SUBAPPLICATION Automatik_Toggle_Button (* Automatik/Hand-Umschalter: 1 VT-Button (latched Toggle) -> Automatik-Zustand als AX-Plug (AUTOMATIK) + dessen Inverses (AX_MAN, fuer PID-Regler MAN-Eingang) + lokaler Publish (ID_AUTOMATIK_STATE_WRITE) fuer VT-Status/Web-Dashboard. Wiederverwendbar fuer jede Automatik-Funktion (Oelkuehler, Aufnahme, ...). *)
  (* Standard: 61499-2; Description: Copyright (c) 2026 Meisterschulen am Ostbahnhof This program and the accompanying materials are made available under the terms of the Eclipse Public License 2.0 which is available at https://www.eclipse.org/legal/epl-2.0/ SPDX-License-Identifier: EPL-2.0 *)
  (* Version 1.12, 2026-09-29, Franz Höpfinger, Meisterschulen am Ostbahnhof, Franz: AUTOMATIK_TOGGLED war falsch benannt/gefiltert - feuerte bei JEDEM Klick, auch beim Ausschalten. Umbenannt in AUTOMATIK_SET_FROM_VT und per neuem E_SWITCH (G=E_T_FF_Automatik.Q VOR dem Klick, ueber AX_SPLIT_4_Automatik auf AX_SPLIT_5 erweitert) gefiltert: EO0 (G=0, AUS->EIN) feuert AUTOMATIK_SET_FROM_VT UND E_T_FF_Automatik.S, EO1 (G=1, EIN->AUS) feuert nur E_T_FF_Automatik.R. CLK jetzt unbenutzt (ersatzlos, S/R decken beide Richtungen ab). *)
  (* Version 1.11, 2026-09-29, Franz Höpfinger, Meisterschulen am Ostbahnhof, Franz: 'Button_Softkey_Aux_IE mergt bereits intern, man kann das Merge rausnehmen' - E_MERGE_Toggle entfernt (Button_Automatik_Toggle ist seit Franz' eigenem Umbau bereits MyLib::sys::Button_Softkey_Aux_IE, das Button/Softkey/Aux selbst zu einem IND zusammenfuehrt; der separate TOGGLE-SubAppEventInput war ohnehin schon unbenutzt/entfernt). Button_Automatik_Toggle.IND geht jetzt direkt auf AX_E_PERMIT_2.EI2. Neuer SubAppEventOutput AUTOMATIK_TOGGLED (von AX_E_PERMIT_2.EO2, also PERMIT-gefiltert) - feuert bei jedem Klick, der die Automatik tatsaechlich toggelt (Button/Softkey/Aux gleichermassen). Fuer Bunker_Ernte_Automatik.SUB: SET soll durch den Display-Klick kommen, nicht durch das FORCE_ON-Echo (Franz-Diagnose: B05-Flattern -> Bunker_Komplett_Absenken.FORCE_ON_OUT -> Befuellautomatik AUTOMATIK-Republish -> Bunker_Ernte_Automatik.ACTIVE wird ueber dieselbe B05-Flanke sofort wieder gesetzt UND resettet, Latch flackert). *)
  (* Version 1.9, 2026-09-27, Franz Höpfinger, Meisterschulen am Ostbahnhof, Franz: 'soll das GESAMTE AN/Aus gaten, beim Uebergang 1->0 einmalig RESET, sonst wirkt es wie ein AX_PERMIT'. Neuer Socket PERMIT (AX). AX_SPLIT_2 speist AX_E_PERMIT_2 (gated FORCE_ON + Button_Automatik_Toggle.IND durch, nur wenn PERMIT=TRUE) und einen neuen AX_F_TRIG (fallende Flanke auf PERMIT -> E_T_FF_Automatik.R). *)
  (* Version 1.8, 2026-09-27, Franz Höpfinger, Meisterschulen am Ostbahnhof, Franz: 'FORCE_ON und FORCE_OFF sollten EVENTS sein, alles andere macht keinen Sinn' - von AX-Sockets (mit internem AX_R_TRIG zur Flankenerkennung) auf echte SubAppEventInputs umgestellt, direkt auf E_T_FF_Automatik.S/.R verdrahtet (wie das bereits bestehende AUS-Event). AX_R_TRIG_ForceOn/_ForceOff entfallen ersatzlos. Aufrufer mit pegelbasierten Quellen (Subscribes, ODER/UND-Verknuepfungen) muessen jetzt selbst die Flankenerkennung vor der Event-Verbindung liefern - siehe Befuellautomatik.SUB/Aufnahme_Automatik.SUB. *)
  (* Version 1.7, 2026-09-20, Franz Höpfinger, Meisterschulen am Ostbahnhof, Bugfix: seit v1.6 (Button_IE statt Softkey_IE, Latchable=0) kommt der Klick zwar an, aber der Button zeigte den AUTOMATIK-Zustand nicht mehr an - bei Latchable=1 hatte das VT dieses Feedback bisher selbst uebernommen (eigene Latched-Optik), das entfaellt jetzt. Neue SubApp Background_Automatik (GreenWhiteBackground3_AX, faerbt Button UND AUX gruen/weiss) ergaenzt, AX_SPLIT_3_Automatik auf AX_SPLIT_4_Automatik erweitert (4. Ausgang -> Background_Automatik.DI1). *)
  (* Version 1.6, 2026-09-20, Franz Höpfinger, Meisterschulen am Ostbahnhof, Bugfix: Button_Automatik_Toggle nutzte Softkey_Aux_IE (Softkey_IE) mit einer echten VT-Button-Object-ID (CButton, z.B. Button_Aufnahme_Geschwindigkeitsregelung_EinAus) - Softkey_IE empfaengt aber keine Button-Activation-Message, der Toggle-Klick kam nie an, AUTOMATIK blieb dauerhaft auf bDefaultAutomatik stehen. Neuer Baustein Button_Aux_IE (Button_IE statt Softkey_IE) - der VT-Button muss dafuer non-latching sein (Latchable=0), wird von Franz direkt im Pool umgestellt. *)
  (* Version 1.5, 2026-09-16, Franz Höpfinger, Meisterschulen am Ostbahnhof, Event-Input RESET in AUS umbenannt (Franz: 'der Eingang soll AUS heissen') - Namenskonsistenz mit AX_SoftkeyToggle_RS_TO_AX(_BG_PUBLISH)/Baender_Individual_Toggle/Baender_EinAus/Aufnahme_Automatik/Ernteseite_Antriebe. *)
  (* Version 1.4, 2026-09-16, Franz Höpfinger, Meisterschulen am Ostbahnhof, Event-Input RESET ergaenzt (rein additiv, zusaetzlich zum bestehenden Reset.IND-Pfad auf E_T_FF_Automatik.R verdrahtet) - fuer einen zentral gelesenen, gemeinsamen SoftKey (z.B. 'Alles Aus'), der mehrere Automatik-Instanzen gleichzeitig per Event zuruecksetzen soll. *)
  (* Version 1.3, 2026-09-15, Franz Höpfinger, Meisterschulen am Ostbahnhof, AUX-Unterstuetzung ergaenzt: Button_Automatik_Toggle von isobus::UT::io::Button::Button_IE (nur SoftKey) auf MyLib::sys::Softkey_Aux_IE (SoftKey ODER AUX) umgestellt, neuer optionaler InputVar u16ObjIdA_Automatik_Toggle (Default ID_NULL) - etabliertes Muster aus AX_SoftkeyToggle_RS_TO_AX.SUB uebernommen. Rein additiv, bestehende Instanzen ohne AUX-Wert funktionieren unveraendert. *)
  (* Version 1.2, 2026-09-13, Franz Höpfinger, Meisterschulen am Ostbahnhof, FORCE_ON/FORCE_OFF Sockets (AX) ergaenzt - rein FB-interne (nicht VT-Objekt-basierte) Gegenstuecke zum bestehenden VT-Reset, je per AX_R_TRIG (steigende Flanke) auf E_T_FF_Automatik.S bzw. .R. Fuer Automatik-zu-Automatik-Verknuepfungen (z.B. Befuellautomatik EIN schaltet Bunker-Ernte-Automatik automatisch mit ein; ein Kollisionsschutz schaltet eine Automatik hart aus) - rein additiv, bestehende Instanzen unveraendert nutzbar. *)
  (* Version 1.1, 2026-09-13, Franz Höpfinger, Meisterschulen am Ostbahnhof, Reset-Eingang ergaenzt (u16ObjId_RESET/u16ObjIdA_RESET/ID_RESET_METHOD -> MyLib::sys::Softkey_Aux_Method_IE -> E_T_FF_Automatik.R), analog AX_SoftkeyToggle_RS_TO_AX - fuer eine globale Sammel-AUS-Taste (SoftKey_AUS), die die Automatik hart auf Hand/AUS zurueckschalten muss (KVE14 Funktionen und Bedingungen Zeile 19, 'Aufnahme, Saege und Baender AUS'). *)
  (* Version 1.0, 2026-09-12, Franz Höpfinger, Meisterschulen am Ostbahnhof, initial implementation - aus Aufnahme_Automatik.SUB herausgeloest (Button_Automatik_Toggle/E_T_FF_Automatik/AX_SPLIT_3_Automatik/AX_NOT_Man/AX_PUBLISH_Automatik), generisch wiederverwendbar. *)
  PACKAGE MyLib::sys;
  IMPORT isobus::UT::Q::const::IDs::ID_NULL;
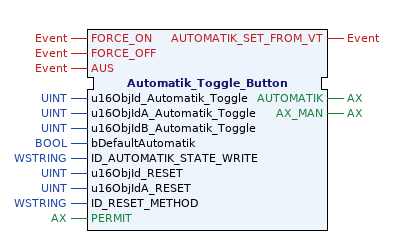
  EVENT_INPUT
    FORCE_ON; (* Schaltet die Automatik hart EIN (z.B. von einer anderen, uebergeordneten Automatik oder einem Methodenaufruf). Unverdrahtet lassen, wenn nicht gebraucht. *)
    FORCE_OFF; (* Schaltet die Automatik hart AUS (z.B. von einem Kollisionsschutz-Methodenaufruf). Unverdrahtet lassen, wenn nicht gebraucht. *)
    AUS; (* Reset hart auf Hand/AUS, von aussen als Event (z.B. 1 zentral gelesener gemeinsamer SoftKey) - zusaetzlich zum eigenen u16ObjId_RESET/u16ObjIdA_RESET/ID_RESET_METHOD-Pfad. Unverdrahtet lassen, wenn nicht gebraucht. *)
  END_EVENT
  EVENT_OUTPUT
    AUTOMATIK_SET_FROM_VT; (* Feuert nur beim Klick (Button/Softkey/Aux, PERMIT-gefiltert), der die Automatik von AUS auf EIN schaltet (per E_SWITCH auf dem Q-Zustand VOR dem Klick gefiltert - ein Klick der AUS schaltet feuert das NICHT). Echter Display-Klick-Event, kein Zustands-Level/Republish. *)
  END_EVENT
  VAR_INPUT
    u16ObjId_Automatik_Toggle : UINT := ID_NULL; (* Object ID VT-Softkey (Automatik/Hand-Umschalter) *)
    u16ObjIdA_Automatik_Toggle : UINT := ID_NULL; (* Object ID AuxFunction2 (Joystick), gleichberechtigt zum VT-Button - optional, ID_NULL wenn kein AUX gebraucht wird *)
    u16ObjIdB_Automatik_Toggle : UINT; (* Object ID VT-Button (Automatik/Hand-Umschalter) *)
    bDefaultAutomatik : BOOL := FALSE; (* Automatik-Zustand beim Start *)
    ID_AUTOMATIK_STATE_WRITE : WSTRING; (* Lokale Publish-Adresse (BOOL, ACTION=WRITE) fuer den Automatik-Ein/Aus-Zustand - Status-Text auf der VT + Web-Client/Dashboard *)
    u16ObjId_RESET : UINT := ID_NULL; (* Object ID Softkey 'Alles Aus' (Reset, hart auf Hand/AUS) - z.B. SoftKey_AUS *)
    u16ObjIdA_RESET : UINT := ID_NULL; (* Object ID AuxFunction2 (Joystick) fuer den Reset - gleichberechtigt zum Softkey 'Alles Aus' *)
    ID_RESET_METHOD : WSTRING; (* Lokale Methodenadresse (ACTION=CREATE_METHOD) fuer den argumentlosen Reset-Trigger (hart auf Hand/AUS) - wird von Web-Client UND OPC-Dashboard aufgerufen *)
  END_VAR
  SOCKETS
    PERMIT : adapter::types::unidirectional::AX;
  END_SOCKETS
  PLUGS
    AUTOMATIK : adapter::types::unidirectional::AX; (* Automatik aktiv (roh, z.B. fuer eine Freigabe-UND-Verknuepfung) *)
    AX_MAN : adapter::types::unidirectional::AX; (* NICHT Automatik aktiv (fuer PID-Regler MAN-Eingang) *)
  END_PLUGS
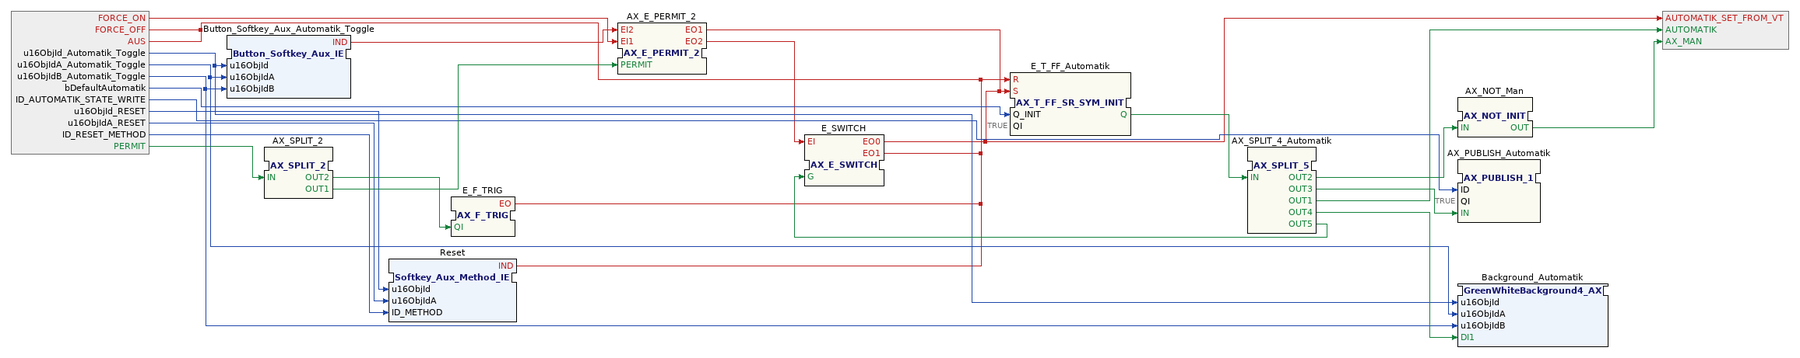
  FBS
    E_T_FF_Automatik : adapter::events::unidirectional::AX_T_FF_SR_SYM_INIT(QI := TRUE);
    AX_SPLIT_4_Automatik : adapter::events::unidirectional::AX_SPLIT_5;
    AX_NOT_Man : adapter::booleanOperators::AX_NOT_INIT;
    AX_PUBLISH_Automatik : adapter::net::AX_PUBLISH_1(QI := TRUE);
    AX_E_PERMIT_2 : adapter::events::unidirectional::AX_E_PERMIT_2;
    AX_SPLIT_2 : adapter::events::unidirectional::AX_SPLIT_2;
    E_F_TRIG : adapter::events::unidirectional::AX_F_TRIG;
    E_SWITCH : adapter::events::unidirectional::AX_E_SWITCH;
  END_FBS
  SUBAPPS
    Button_Softkey_Aux_Automatik_Toggle : MyLib::sys::Button_Softkey_Aux_IE;
    Background_Automatik : MyLib::sys::GreenWhiteBackground4_AX;
    Reset : MyLib::sys::Softkey_Aux_Method_IE;
  END_SUBAPPS
  EVENT_CONNECTIONS
    Button_Softkey_Aux_Automatik_Toggle.IND TO AX_E_PERMIT_2.EI2;
    Reset.IND TO E_T_FF_Automatik.R;
    AUS TO E_T_FF_Automatik.R;
    FORCE_ON TO AX_E_PERMIT_2.EI1;
    FORCE_OFF TO E_T_FF_Automatik.R;
    AX_E_PERMIT_2.EO1 TO E_T_FF_Automatik.S;
    AX_E_PERMIT_2.EO2 TO E_SWITCH.EI;
    E_SWITCH.EO0 TO AUTOMATIK_SET_FROM_VT;
    E_F_TRIG.EO TO E_T_FF_Automatik.R;
    E_SWITCH.EO0 TO E_T_FF_Automatik.S;
    E_SWITCH.EO1 TO E_T_FF_Automatik.R;
  END_CONNECTIONS
  DATA_CONNECTIONS
    u16ObjId_Automatik_Toggle TO Button_Softkey_Aux_Automatik_Toggle.u16ObjId;
    u16ObjIdA_Automatik_Toggle TO Button_Softkey_Aux_Automatik_Toggle.u16ObjIdA;
    u16ObjId_Automatik_Toggle TO Background_Automatik.u16ObjId;
    u16ObjIdA_Automatik_Toggle TO Background_Automatik.u16ObjIdA;
    bDefaultAutomatik TO E_T_FF_Automatik.Q_INIT;
    ID_AUTOMATIK_STATE_WRITE TO AX_PUBLISH_Automatik.ID;
    u16ObjId_RESET TO Reset.u16ObjId;
    u16ObjIdA_RESET TO Reset.u16ObjIdA;
    ID_RESET_METHOD TO Reset.ID_METHOD;
    u16ObjIdB_Automatik_Toggle TO Button_Softkey_Aux_Automatik_Toggle.u16ObjIdB;
    u16ObjIdB_Automatik_Toggle TO Background_Automatik.u16ObjIdB;
  END_CONNECTIONS
  ADAPTER_CONNECTIONS
    E_T_FF_Automatik.Q TO AX_SPLIT_4_Automatik.IN;
    AX_SPLIT_4_Automatik.OUT2 TO AX_NOT_Man.IN;
    AX_SPLIT_4_Automatik.OUT3 TO AX_PUBLISH_Automatik.IN;
    AX_NOT_Man.OUT TO AX_MAN;
    AX_SPLIT_4_Automatik.OUT1 TO AUTOMATIK;
    AX_SPLIT_4_Automatik.OUT4 TO Background_Automatik.DI1;
    PERMIT TO AX_SPLIT_2.IN;
    AX_SPLIT_2.OUT2 TO E_F_TRIG.QI;
    AX_SPLIT_2.OUT1 TO AX_E_PERMIT_2.PERMIT;
    AX_SPLIT_4_Automatik.OUT5 TO E_SWITCH.G;
  END_CONNECTIONS
END_SUBAPPLICATION
